FUNCTION_BLOCK FB_WriteRFIDnew
VAR_INPUT
	bAutoNumber				:BOOL;		
	byFirstByteInput		:BYTE;
	bySecondByteInput		:BYTE;
	byLastByteInput			:BYTE;

	bReset					:BOOL;		//reset licznika
END_VAR
VAR_IN_OUT
	bEnable					:BOOL;		//zalczenie bloku
	byIDtoWrite				:BYTE;		//ID do wczytania
END_VAR


VAR_OUTPUT
	byFirstByteOutput		:BYTE;
	bySecondByteOutput		:BYTE;
	byThirdByteOutput		:BYTE;
	byFourthByteOutput		:BYTE;
	byFifthByteOutput		:BYTE;
	byLastByteOutput		:BYTE;
	bDone					:BOOL;		//informacja o prawidlowym zakoczeniu zapisu
	bError					:BOOL;
	iCounterDone			:INT;		//licznik operacji zapisu zakonczonych sukcesem
END_VAR
VAR
	
	iStep: INT;
	tonDelayError	:TON;
	tonStep0: TON;
	nAutoNumberCount2: INT;
END_VAR

IF bReset THEN
	iCounterDone	:=0;
	iStep := 0;
	byFirstByteOutput := byLastByteOutput := 0;
	bReset := FALSE;
	nAutoNumberCount2:=0;
END_IF

tonStep0(IN:=iStep=0 AND bEnable,PT:=T#500MS);

CASE iStep OF
	0:  //init	
		IF byFirstByteInput = 129 AND tonStep0.Q THEN
			bDone:=FALSE; 
			iStep:=10;
		END_IF
	
	10:  //write command
		bySecondByteOutput 	:= 02;
		byThirdByteOutput	:= 00;
		byFourthByteOutput	:= 00;
		byFifthByteOutput 	:= 01;
		byFirstByteOutput := byLastByteOutput := 01;
	
		IF byFirstByteInput = 163 THEN
			iStep := 20;
		ELSIF NOT byFirstByteInput = 163 AND tonDelayError.Q = TRUE THEN
			iStep := 100;
		END_IF
	
	20: //write data
	
		bySecondByteOutput := byIDtoWrite;
		
		byFirstByteOutput := byLastByteOutput := 65;
		IF byFirstByteInput = 167 THEN
			iStep := 30;
		ELSIF NOT byFirstByteInput = 167 AND tonDelayError.Q = TRUE THEN
			iStep := 100;
		END_IF
	
	30: //check status
		byFirstByteOutput := byLastByteOutput := 0;
		iCounterDone	:= iCounterDone + 1; 
		bDone			:= TRUE; 	
		IF byFirstByteInput = 128 THEN
			iStep := 0;			
			//Liczenie do dwóch i dopiero potem dodaje +1	
			nAutoNumberCount2 := nAutoNumberCount2 + 1;
			IF nAutoNumberCount2 = 2 THEN
				byIDtoWrite			:= byIDtoWrite+1;
				bEnable				:= FALSE;
				nAutoNumberCount2 	:= 0;
			END_IF
			
		ELSIF NOT byFirstByteInput = 128 AND tonDelayError.Q = TRUE THEN
			iStep := 100;
		END_IF
		
	100: // errors
		bError		:= TRUE;
		



END_CASE

END_FUNCTION_BLOCK

(* stored: Version 1.1.0.1, ProductVersion 3.1.4026.13, FileIdentifier 53ec9395777c9612d9be7c55ae0ef13f6e235981, FileSignature 4508cacae67c7f7c7955e51963f15ac3dc0f34b8dc1c2907b316075552bffd58c995e2740c8587e8dd672e3327e4875434aa8f433040e2b8f8b23e07de02ba6d3ad1404043b0a805f965288bb4fee1e099241f7f978dc6951045649f7f154494c7cfc0c94ce23f5c4df7568f7d6b9a8fe5a4e735b962dbbdbef3deaedcf6c10b1473f8235bbb57e2d734f92851278c1e5f610b6baf2a63ad51da118c4efa612e5ec617c4d214b79dc8ffc38c5c0ff775df903c3e736d024651e87ac675e1d3761a16c5dd646464e05e0e3b83c0c2e73d7795f8c49fc6210765bf9da1666f754a9a6a263494405b633bf6b3a04cd6bcff33eebe9c8e28a767b7c3a248080d4d56
   POU FB_WriteRFIDnew: Id {4d71942d-667c-4b3d-808e-49638e3ce88f}, SpecialFunc None *)
